INTERFACE ITF_TopElement1_HMI_Connector_Command EXTENDS ITF_BaseTopElement_HMI_Connector_Command

END_INTERFACE

(* stored: Version 1.1.0.1
   Itf ITF_TopElement1_HMI_Connector_Command: Id {d6f5eecc-0706-0804-0b62-31b39ad6604f} *)
